// SIMATIC S7-200 project (STEP 7-Micro/WIN), CPU 224 REL 01.22

SYMBOL_TABLE S7-200 Symbols
Always_On        SM0.0    // Always ON
END_SYMBOL_TABLE

SYMBOL_TABLE USR2
Year             VB0      // Year (00-99)
Month            VB1      // Month (01-12)
Day              VB2      // Day (01-31)
Hour             VB3      // Hour (00-23)
Minute           VB4      // Minute (00-59)
Second           VB5      // Second (00-59)
Weekday          VB7      // Day Of Week (0-Disable, 1-Sunday, 7-Saturday)
WYear            VB10
WMonth           VB11
WDay             VB12
WHour            VB13
WMinute          VB14
WSecond          VB15
WWeekday         VB17
ClockAhead       M0.0
ClockBack        M0.1
ClockBackNoRepeat M0.2
END_SYMBOL_TABLE

ORGANIZATION_BLOCK MAIN:OB1
TITLE=This project includes a Daylight Savings Time (DST) automatic adjustment module, implementing automatic DST adjustment for the internal clock of the Siemens S7-200 PLC. The controlled device is the PLC's internal clock, suitable for scenarios such as production scheduling and data logging.
// When the program runs, it first reads the current year, month, date, hour, and day of the week from the PLC's real-time clock to provide data for subsequent judgments.
// In April each year, when the current month is April, the day of the week is Sunday, the date is between 1 and 7, and the hour is 2 AM, the program determines it is time to advance the clock and sets the clock-ahead flag.
// At this point, the system copies the current time to the write addresses for the year and other fields, increments the write hour value (from 2 AM to 3 AM), and writes the adjusted time to the real-time clock, ensuring the time is advanced by one hour.
// Similarly, in October each year, when the current month is October, the day of the week is Sunday, the date is between 25 and 31, and the hour is 2 AM, the program sets the clock-back flag.
// If the clock-back repeat prevention flag is not set, the system copies the current time to the write addresses for the year and other fields, decrements the write hour value (from 2 AM to 1 AM), writes the adjusted time, and immediately sets the clock-back repeat prevention flag.
// This prevents the clock-back operation from being repeated due to program loops, ensuring the time is adjusted only once.
// Subsequently, when the current hour reaches 3 AM, the clock-back repeat prevention flag is reset, preparing for the next DST adjustment.
// During the time adjustment, the write hour value changes based on increment or decrement operations, and the system relies on the PLC's built-in mechanisms to prevent time write failures.
BEGIN
Network 1 // Network Title
// Read the real time clock into VB0 thru VB7
LD     Always_On:SM0.0
TODR   Year:VB0
?000
Network 2
// The first Sunday of April at 2AM is when the clocks are to be set ahead one hour.
// Verify the month is April, the weekday is Sunday, the Day is between 1 and 7, and the time is 2AM
LDB=   Month:VB1, 4
AB=    Weekday:VB7, 1
AB>=   Day:VB2, 1
AB<=   Day:VB2, 7
AB=    Hour:VB3, 2
=      ClockAhead:M0.0
Network 3
// When the above criteria is met, it is time to advance the clock one hour.
// Move existing read values to write area.
// Increment Hour.
// Write to real time clock.
LD     ClockAhead:M0.0
EU
BMB    Year:VB0, WYear:VB10, 8
INCB   WHour:VB13
TODW   WYear:VB10
Network 4
// The last Sunday in October at 2AM is when the clock is to be set back one hour.
// Verify the month is October, the weekday is Sunday, the day is between 25 and 31, and the time is 2AM
LDB=   Month:VB1, 10
AB=    Weekday:VB7, 1
AB>=   Day:VB2, 25
AB<=   Day:VB2, 31
AB=    Hour:VB3, 2
=      ClockBack:M0.1
Network 5
// When the above criteria is met, it is time to reverse the clock one hour.
// Move existing read values to write area.
// Decrement Hour.
// Write to real time clock.
// Set a bit so it only happens once.
LD     ClockBack:M0.1
AN     ClockBackNoRepeat:M0.2
EU
BMB    Year:VB0, WYear:VB10, 8
DECB   WHour:VB13
TODW   WYear:VB10
S      ClockBackNoRepeat:M0.2, 1
Network 6
// If the clock has been set back and then reaches 3AM, reset the temporary bit we used above.
LD     ClockBackNoRepeat:M0.2
AB=    Hour:VB3, 3
R      ClockBackNoRepeat:M0.2, 1
END_ORGANIZATION_BLOCK
